TYPE Tank_Io :
STRUCT
	in			: Tank_Io_In;
	out			: Tank_Io_Out;
END_STRUCT
END_TYPE

(* stored: Version 1.1.0.1
   DUT Tank_Io: Id {bd29f8b0-6451-4caa-afdf-62ce3a6deee2} *)
